TYPE ST_UserMgmtHistoryEvent :
STRUCT
    bExecute            : BOOL;

    sTargetUser         : STRING(100);
    sEventType          : STRING(50);

    sOldGroup           : STRING(100);
    sNewGroup           : STRING(100);

    iOldAutoLogoutMin   : INT;
    iNewAutoLogoutMin   : INT;

    sPerformedBy        : STRING(100);
    sSourceScreen       : STRING(100);
    sEventComment       : STRING(255);

    bBusy               : BOOL;
    bDone               : BOOL;
    bError              : BOOL;
    sErrorText          : STRING(255);
END_STRUCT
END_TYPE

(* stored: Version 1.1.0.1, ProductVersion 3.1.4024.15
   DUT ST_UserMgmtHistoryEvent: Id {f88f700f-5dd5-4063-852c-493a937c5c41} *)
